{attribute 'GeneratedUsingTerminal: EJ7037-0000-0020'}
{attribute addProperty BoxType "EJ7037-0000-0020"}
{attribute addProperty Id "EnableBOOL1ResetBOOL1Reduce_torqueBOOL1Digital_output_1BOOL1"}
{attribute addProperty CRC "1607755581"}
{attribute addProperty Size "4"}
TYPE Control_5FD4673D :
STRUCT
	{attribute addProperty Name "Enable"}
	Enable : BOOL;
	{attribute addProperty Name "Reset"}
	Reset : BOOL;
	{attribute addProperty Name "Reduce_torque"}
	Reduce_torque : BOOL;
	{attribute addProperty Name "Digital_output_1"}
	Digital_output_1 : BOOL;
END_STRUCT
END_TYPE
